// Mitsubishi GX Works2 project: LRI - inclusão de SET   PLC: Q03UDV
// HelloWorld

PROGRAM MAIN
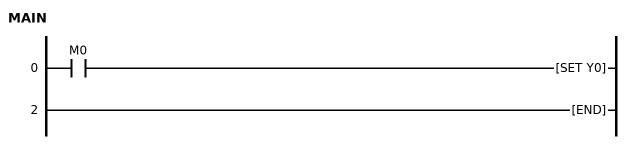
0     LD      M0
      SET     Y0
2     END
END_PROGRAM
